// TIA Portal V20 export
TYPE "s_zc_CellInterlocks"
// stored: Access Published, IsFailsafeCompliant true, Namespace Safety
   STRUCT
      NoEStop { ExternalWritable := 'False'} : Bool := FALSE;   // Estop push button is released and Estop status function is reset (Acknowledged).
      EStopResetReq { ExternalWritable := 'False'} : Bool := FALSE;   // Request the reset ack. from/to other stations.
      AllGatesLocked { ExternalWritable := 'False'} : Bool := FALSE;   // Entire gates are locked on station.
      AllGatesResetReq { ExternalWritable := 'False'} : Bool := FALSE;   // Door is closed and door status function is reset (Acknowledged).
      AnySafetyGatesUnlocked { ExternalWritable := 'False'} : Bool := FALSE;   // Any gate is unlocked or opened on station
      GuardsOK { ExternalWritable := 'False'} : Bool := FALSE;   // Guard Ok will be active both gate and perimeter guarding are reset
      PressSafetyOn { ExternalWritable := 'False'} : Bool := FALSE;   // TBD
      PressSafetyOff { ExternalWritable := 'False'} : Bool := FALSE;   // TBD
      ScrapDoorsClosed { ExternalWritable := 'False'} : Bool := FALSE;   // The NG Box is closed.
      ShutterDoorClosed { ExternalWritable := 'False'} : Bool := FALSE;   // Upper shutter door is closed.
      ShutterDoorOpened { ExternalWritable := 'False'} : Bool := FALSE;   // Upper shutter door is opened.
      LightCurtainNOK { ExternalWritable := 'False'} : Bool := FALSE;   // Light curtain is working and no interference.
      LightCurtainMunting { ExternalWritable := 'False'} : Bool := FALSE;   // Light curtain function is muting.
      anodeConveyorCoversOK { ExternalWritable := 'False'} : Bool;   // Conveyor Cover Closed
      cathodeConveyorCoversOK { ExternalWritable := 'False'} : Bool;   // Conveyor Cover Closed
      ConveyorCoversSystemFaults { ExternalWritable := 'False'} : Bool;   // Safety Cards System Faults
   END_STRUCT;
END_TYPE
